# EPICS autosave request: 100idPyCRLApp/Db/pyDevCRL_stack_move_settings.req
file sseqRecord_settings.req P=$(P)$(SYSID):$(OE):,S=stack$(M)_move
file scalcout_settings.req P=$(P)$(SYSID):$(OE):stack$(M)_RBV_calc
